FUNCTION_BLOCK ConveyorControllerIProv (* Conveyor Controller Interface Provider *)
  (* Standard: 61499-2 *)
  (* Version 0.2, 2003-12-05, JHC, Rockwell Automation, Renamed from NEWCOMPFB. *)
  (* Version 0.1, 2002-01-08, JHC, Rockwell Automation, Added DLY FB as example. *)
  (* Version 0.0, 2000-05-27, JHC, Rockwell Automation *)
  (* Compiler header: package fb.rt.dasdA1.A2.Conveyor; *)
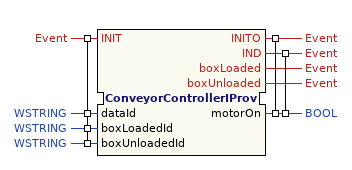
  EVENT_INPUT
    INIT WITH dataId, boxLoadedId, boxUnloadedId; (* Initialization Request *)
  END_EVENT
  EVENT_OUTPUT
    INITO WITH motorOn; (* Initialization Confirm *)
    IND WITH motorOn;
    boxLoaded;
    boxUnloaded;
  END_EVENT
  VAR_INPUT
    dataId : WSTRING;
    boxLoadedId : WSTRING;
    boxUnloadedId : WSTRING;
  END_VAR
  VAR_OUTPUT
    motorOn : BOOL;
  END_VAR
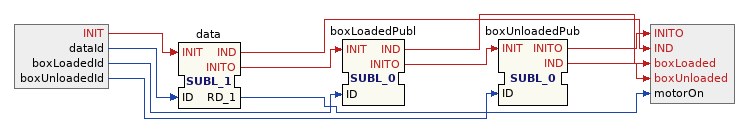
  FBS
    data : SUBL_1;
    boxLoadedPubl : SUBL_0;
    boxUnloadedPub : SUBL_0;
  END_FBS
  EVENT_CONNECTIONS
    INIT TO data.INIT;
    data.IND TO IND;
    data.INITO TO boxLoadedPubl.INIT;
    boxLoadedPubl.IND TO boxLoaded;
    boxLoadedPubl.INITO TO boxUnloadedPub.INIT;
    boxUnloadedPub.INITO TO INITO;
    boxUnloadedPub.IND TO boxUnloaded;
  END_CONNECTIONS
  DATA_CONNECTIONS
    dataId TO data.ID;
    boxLoadedId TO boxLoadedPubl.ID;
    data.RD_1 TO motorOn;
    boxUnloadedId TO boxUnloadedPub.ID;
  END_CONNECTIONS
END_FUNCTION_BLOCK
